// TIA Portal project "Entrega1 automatas2" (V17)

(* hardware
DEVICE "S7-1200 station_1"  S7-1200 Station
   slot 0: "Rack_0"  S7-1200 Rack  Rack  V1.0
   slot 1: "PLC_1"  CPU 1215C AC/DC/Rly  6ES7 215-1BG40-0XB0  V4.0
DEVICE "S7-1200 station_2"  S7-1200 Station
   slot 0: "Rack_0"  S7-1200 Rack  Rack  V1.0
   slot 1: "PLC_2"  CPU 1214C AC/DC/Rly  6ES7 214-1BG31-0XB0  V3.0
   slot 3: "AQ 1x12BIT_1"  AQ1 signal board  6ES7 232-4HA30-0XB0  V1.0
DEVICE "S7-1200 station_3"  S7-1200 Station
   slot 0: "Rack_0"  S7-1200 Rack  Rack  V1.0
   slot 1: "PLC_3"  CPU 1214C AC/DC/Rly  6ES7 214-1BG31-0XB0  V3.0
*)

// ===== PLC "PLC_1"  CPU 1215C AC/DC/Rly =====

VAR_GLOBAL   // PLC tag table "Default tag table"
   "i_PM" AT %I0.0 : Bool;
   "i_PP" AT %I0.1 : Bool;
   "i_FC" AT %I0.2 : Bool;
   "q_EV1" AT %Q0.0 : Bool;
   "q_EV2" AT %Q0.1 : Bool;
   "q_EV3" AT %Q0.2 : Bool;
   "q_Di1" AT %Q0.3 : Bool;
   "q_Di2" AT %Q0.4 : Bool;
   "q_Z" AT %Q0.5 : Bool;
   "q_KM1" AT %Q0.6 : Bool;
   "q_KM2" AT %Q0.7 : Bool;
   "GP_E0" AT %M50.0 : Bool;
   "GP_E1" AT %M50.1 : Bool;
   "GP_E2" AT %M50.2 : Bool;
   "GP_E3" AT %M50.3 : Bool;
   "GP_E4" AT %M50.4 : Bool;
   "GP_E5" AT %M50.5 : Bool;
   "GP_E6" AT %M50.6 : Bool;
   "GP_E7" AT %M50.7 : Bool;
   "GS_E100" AT %M51.0 : Bool;
   "GS_E101" AT %M51.1 : Bool;
   "T1" AT %MD100 : Time;
   "Minimo_distancia" AT %MD104 : Real;
   "Maximo distancia" AT %MD106 : Real;
   "Salida_Voltios" AT %MD80 : Real;
   "distancia_normalizada" AT %MD60 : Real;
   "Variable_Stop" AT %M500.0 : Bool;
END_VAR

VAR_GLOBAL   // PLC tag table "Tag table_1"
   "entrada_analogica(1)" AT %IW64 : Word;
END_VAR

// folder: System blocks/Program resources

DATA_BLOCK "T1.1"   // DB1
{ S7_Optimized_Access := 'TRUE' }
AUTHOR : Simatic
FAMILY : IEC
NAME : IEC_TMR
VERSION : 1.0
// stored: InstanceOfName IEC_TIMER
"IEC_TIMER"
BEGIN
END_DATA_BLOCK

DATA_BLOCK "T2"   // DB2
{ S7_Optimized_Access := 'TRUE' }
AUTHOR : Simatic
FAMILY : IEC
NAME : IEC_TMR
VERSION : 1.0
// stored: InstanceOfName IEC_TIMER
"IEC_TIMER"
BEGIN
END_DATA_BLOCK

DATA_BLOCK "T3"   // DB3
{ S7_Optimized_Access := 'TRUE' }
AUTHOR : Simatic
FAMILY : IEC
NAME : IEC_TMR
VERSION : 1.0
// stored: InstanceOfName IEC_TIMER
"IEC_TIMER"
BEGIN
END_DATA_BLOCK

DATA_BLOCK "T4"   // DB4
{ S7_Optimized_Access := 'TRUE' }
AUTHOR : Simatic
FAMILY : IEC
NAME : IEC_TMR
VERSION : 1.0
// stored: InstanceOfName IEC_TIMER
"IEC_TIMER"
BEGIN
END_DATA_BLOCK

// folder: (top level)

FUNCTION "Grafcet principal" : Void   // FC1, LAD
{ S7_Optimized_Access := 'TRUE' }
VERSION : 0.1
   VAR_TEMP   // added for the SCL form of the ladder/FBD networks
      _w1 : Bool;
   END_VAR
BEGIN

REGION Network 1
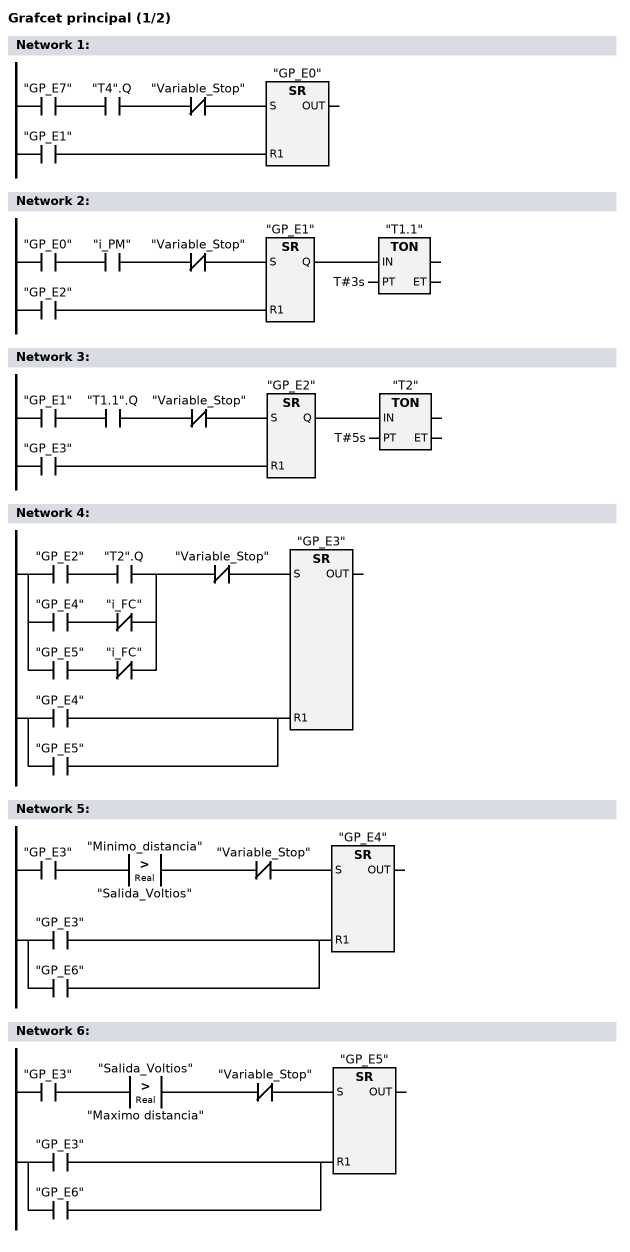
   RUNG wire#powerrail
      Contact( "GP_E7" )
      Contact( "T4".Q )
      I_Contact( "Variable_Stop" )
      S_SR(operand := "GP_E0", r1 := wire#w1)
   END_RUNG
   RUNG wire#powerrail
      Contact( "GP_E1" )
   END_RUNG wire#w1
   // the same network as SCL:
   IF "GP_E7" AND "T4".Q AND NOT "Variable_Stop" THEN
       "GP_E0" := TRUE;   // SR flip-flop
   END_IF;
   IF "GP_E1" THEN "GP_E0" := FALSE; END_IF;
END_REGION

REGION Network 2
   IF "GP_E0" AND "i_PM" AND NOT "Variable_Stop" THEN
       "GP_E1" := TRUE;   // SR flip-flop
   END_IF;
   IF "GP_E2" THEN "GP_E1" := FALSE; END_IF;
   "T1.1".TON(IN := "GP_E1", PT := T#3s);
END_REGION

REGION Network 3
   IF "GP_E1" AND "T1.1".Q AND NOT "Variable_Stop" THEN
       "GP_E2" := TRUE;   // SR flip-flop
   END_IF;
   IF "GP_E3" THEN "GP_E2" := FALSE; END_IF;
   "T2".TON(IN := "GP_E2", PT := T#5s);
END_REGION

REGION Network 4
   RUNG wire#powerrail
      Contact( "GP_E2" )
      Contact( "T2".Q )
      wire#w1
      I_Contact( "Variable_Stop" )
      S_SR(operand := "GP_E3", r1 := wire#w2)
   END_RUNG
   RUNG wire#powerrail
      Contact( "GP_E4" )
      I_Contact( "i_FC" )
   END_RUNG wire#w1
   RUNG wire#powerrail
      Contact( "GP_E5" )
      I_Contact( "i_FC" )
   END_RUNG wire#w1
   RUNG wire#powerrail
      Contact( "GP_E4" )
   END_RUNG wire#w2
   RUNG wire#powerrail
      Contact( "GP_E5" )
   END_RUNG wire#w2
   // the same network as SCL:
   IF (("GP_E2" AND "T2".Q) OR ("GP_E4" AND NOT "i_FC") OR ("GP_E5" AND NOT "i_FC")) AND NOT "Variable_Stop" THEN
       "GP_E3" := TRUE;   // SR flip-flop
   END_IF;
   IF "GP_E4" OR "GP_E5" THEN "GP_E3" := FALSE; END_IF;
END_REGION

REGION Network 5
   RUNG wire#powerrail
      Contact( "GP_E3" )
      { S7_Templates := "SrcType := Real" } GT_Contact(in1 := "Minimo_distancia", in2 := "Salida_Voltios")
      I_Contact( "Variable_Stop" )
      S_SR(operand := "GP_E4", r1 := wire#w1)
   END_RUNG
   RUNG wire#powerrail
      Contact( "GP_E3" )
   END_RUNG wire#w1
   RUNG wire#powerrail
      Contact( "GP_E6" )
   END_RUNG wire#w1
   // the same network as SCL:
   IF "GP_E3" AND ("Minimo_distancia" > "Salida_Voltios") AND NOT "Variable_Stop" THEN
       "GP_E4" := TRUE;   // SR flip-flop
   END_IF;
   IF "GP_E3" OR "GP_E6" THEN "GP_E4" := FALSE; END_IF;
END_REGION

REGION Network 6
   RUNG wire#powerrail
      Contact( "GP_E3" )
      { S7_Templates := "SrcType := Real" } GT_Contact(in1 := "Salida_Voltios", in2 := "Maximo distancia")
      I_Contact( "Variable_Stop" )
      S_SR(operand := "GP_E5", r1 := wire#w1)
   END_RUNG
   RUNG wire#powerrail
      Contact( "GP_E3" )
   END_RUNG wire#w1
   RUNG wire#powerrail
      Contact( "GP_E6" )
   END_RUNG wire#w1
   // the same network as SCL:
   IF "GP_E3" AND ("Salida_Voltios" > "Maximo distancia") AND NOT "Variable_Stop" THEN
       "GP_E5" := TRUE;   // SR flip-flop
   END_IF;
   IF "GP_E3" OR "GP_E6" THEN "GP_E5" := FALSE; END_IF;
END_REGION

REGION Network 7
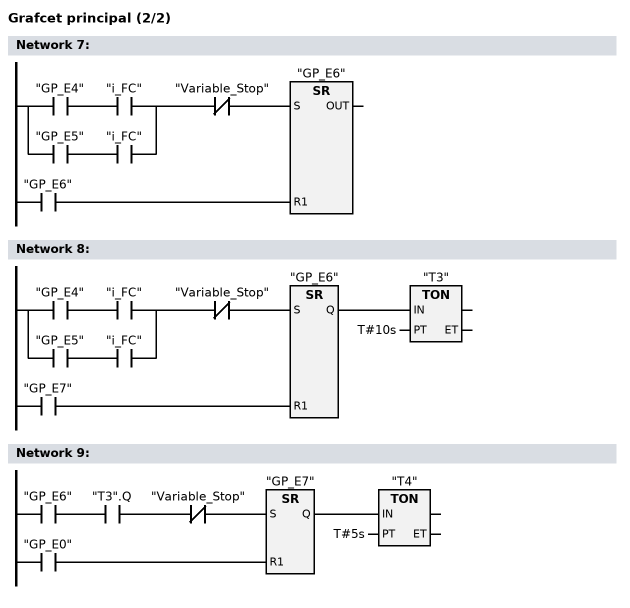
   RUNG wire#powerrail
      Contact( "GP_E4" )
      Contact( "i_FC" )
      wire#w1
      I_Contact( "Variable_Stop" )
      S_SR(operand := "GP_E6", r1 := wire#w2)
   END_RUNG
   RUNG wire#powerrail
      Contact( "GP_E5" )
      Contact( "i_FC" )
   END_RUNG wire#w1
   RUNG wire#powerrail
      Contact( "GP_E6" )
   END_RUNG wire#w2
   // the same network as SCL:
   #_w1 := "GP_E6";
   IF (("GP_E4" AND "i_FC") OR ("GP_E5" AND "i_FC")) AND NOT "Variable_Stop" THEN
       "GP_E6" := TRUE;   // SR flip-flop
   END_IF;
   IF #_w1 THEN "GP_E6" := FALSE; END_IF;
END_REGION

REGION Network 8
   IF (("GP_E4" AND "i_FC") OR ("GP_E5" AND "i_FC")) AND NOT "Variable_Stop" THEN
       "GP_E6" := TRUE;   // SR flip-flop
   END_IF;
   IF "GP_E7" THEN "GP_E6" := FALSE; END_IF;
   "T3".TON(IN := "GP_E6", PT := T#10s);
END_REGION

REGION Network 9
   IF "GP_E6" AND "T3".Q AND NOT "Variable_Stop" THEN
       "GP_E7" := TRUE;   // SR flip-flop
   END_IF;
   IF "GP_E0" THEN "GP_E7" := FALSE; END_IF;
   "T4".TON(IN := "GP_E7", PT := T#5s);
END_REGION
END_FUNCTION

FUNCTION "Grafcet Stop" : Void   // FC2, LAD
{ S7_Optimized_Access := 'TRUE' }
VERSION : 0.1
BEGIN

REGION Network 1
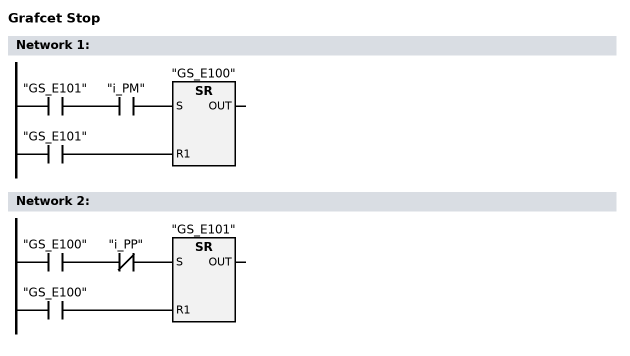
   RUNG wire#powerrail
      Contact( "GS_E101" )
      Contact( "i_PM" )
      S_SR(operand := "GS_E100", r1 := wire#w1)
   END_RUNG
   RUNG wire#powerrail
      Contact( "GS_E101" )
   END_RUNG wire#w1
   // the same network as SCL:
   IF "GS_E101" AND "i_PM" THEN
       "GS_E100" := TRUE;   // SR flip-flop
   END_IF;
   IF "GS_E101" THEN "GS_E100" := FALSE; END_IF;
END_REGION

REGION Network 2
   RUNG wire#powerrail
      Contact( "GS_E100" )
      I_Contact( "i_PP" )
      S_SR(operand := "GS_E101", r1 := wire#w1)
   END_RUNG
   RUNG wire#powerrail
      Contact( "GS_E100" )
   END_RUNG wire#w1
   // the same network as SCL:
   IF "GS_E100" AND NOT "i_PP" THEN
       "GS_E101" := TRUE;   // SR flip-flop
   END_IF;
   IF "GS_E100" THEN "GS_E101" := FALSE; END_IF;
END_REGION
END_FUNCTION

FUNCTION "Salidas" : Void   // FC3, LAD
{ S7_Optimized_Access := 'TRUE' }
VERSION : 0.1
BEGIN

REGION Network 1
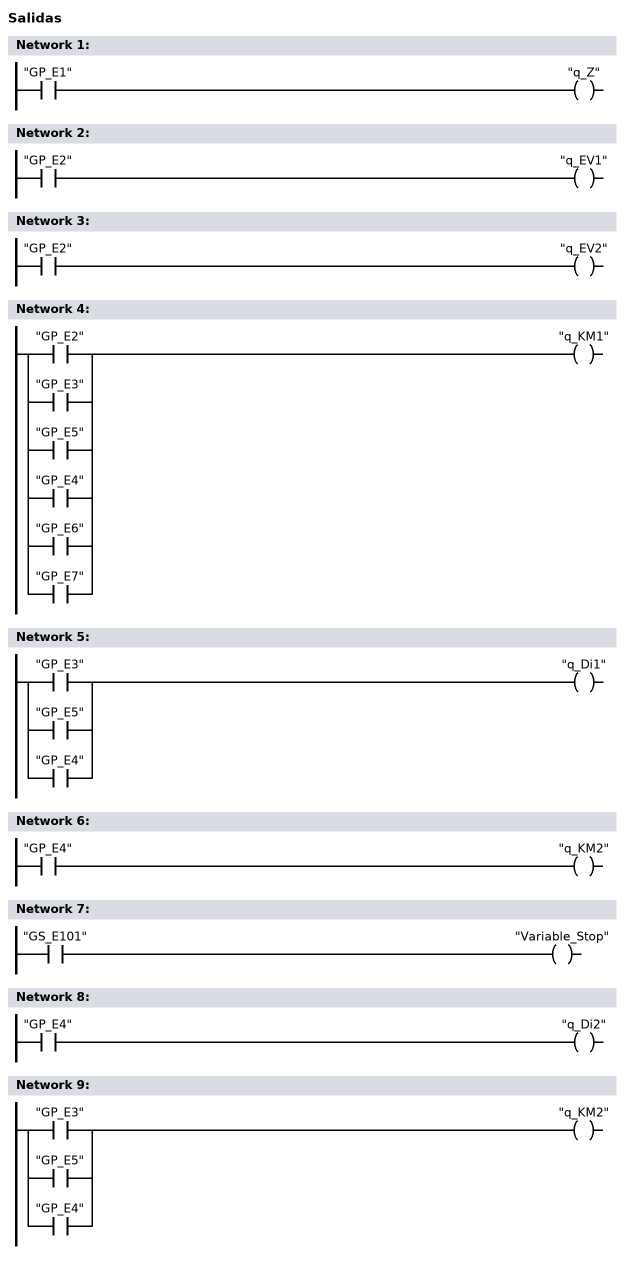
   RUNG wire#powerrail
      Contact( "GP_E1" )
      Coil( "q_Z" )
   END_RUNG
   // the same network as SCL:
   "q_Z" := "GP_E1";
END_REGION

REGION Network 2
   RUNG wire#powerrail
      Contact( "GP_E2" )
      Coil( "q_EV1" )
   END_RUNG
   // the same network as SCL:
   "q_EV1" := "GP_E2";
END_REGION

REGION Network 3
   RUNG wire#powerrail
      Contact( "GP_E2" )
      Coil( "q_EV2" )
   END_RUNG
   // the same network as SCL:
   "q_EV2" := "GP_E2";
END_REGION

REGION Network 4
   RUNG wire#powerrail
      Contact( "GP_E2" )
      wire#w1
      Coil( "q_KM1" )
   END_RUNG
   RUNG wire#powerrail
      Contact( "GP_E3" )
   END_RUNG wire#w1
   RUNG wire#powerrail
      Contact( "GP_E5" )
   END_RUNG wire#w1
   RUNG wire#powerrail
      Contact( "GP_E4" )
   END_RUNG wire#w1
   RUNG wire#powerrail
      Contact( "GP_E6" )
   END_RUNG wire#w1
   RUNG wire#powerrail
      Contact( "GP_E7" )
   END_RUNG wire#w1
   // the same network as SCL:
   "q_KM1" := "GP_E2" OR "GP_E3" OR "GP_E5" OR "GP_E4" OR "GP_E6" OR "GP_E7";
END_REGION

REGION Network 5
   RUNG wire#powerrail
      Contact( "GP_E3" )
      wire#w1
      Coil( "q_Di1" )
   END_RUNG
   RUNG wire#powerrail
      Contact( "GP_E5" )
   END_RUNG wire#w1
   RUNG wire#powerrail
      Contact( "GP_E4" )
   END_RUNG wire#w1
   // the same network as SCL:
   "q_Di1" := "GP_E3" OR "GP_E5" OR "GP_E4";
END_REGION

REGION Network 6
   RUNG wire#powerrail
      Contact( "GP_E4" )
      Coil( "q_KM2" )
   END_RUNG
   // the same network as SCL:
   "q_KM2" := "GP_E4";
END_REGION

REGION Network 7
   RUNG wire#powerrail
      Contact( "GS_E101" )
      Coil( "Variable_Stop" )
   END_RUNG
   // the same network as SCL:
   "Variable_Stop" := "GS_E101";
END_REGION

REGION Network 8
   RUNG wire#powerrail
      Contact( "GP_E4" )
      Coil( "q_Di2" )
   END_RUNG
   // the same network as SCL:
   "q_Di2" := "GP_E4";
END_REGION

REGION Network 9
   RUNG wire#powerrail
      Contact( "GP_E3" )
      wire#w1
      Coil( "q_KM2" )
   END_RUNG
   RUNG wire#powerrail
      Contact( "GP_E5" )
   END_RUNG wire#w1
   RUNG wire#powerrail
      Contact( "GP_E4" )
   END_RUNG wire#w1
   // the same network as SCL:
   "q_KM2" := "GP_E3" OR "GP_E5" OR "GP_E4";
END_REGION
END_FUNCTION

FUNCTION "Analogicas" : Void   // FC4, LAD
{ S7_Optimized_Access := 'TRUE' }
VERSION : 0.1
BEGIN

REGION Network 1
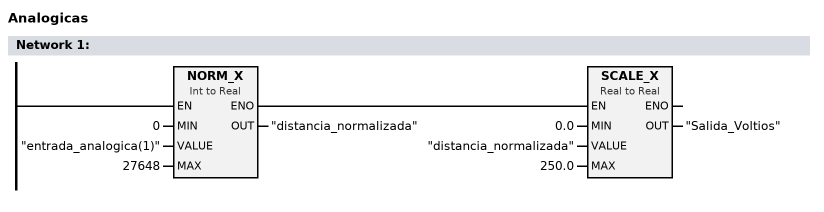
   RUNG wire#powerrail
      { S7_Templates := "[SrcType := Int, DestType := Real]" } Normalize(min := 0, value := "entrada_analogica(1)", max := 27648, out => "distancia_normalizada")
      { S7_Templates := "[SrcType := Real, DestType := Real]" } Scale(min := 0.0, value := "distancia_normalizada", max := 250.0, out => "Salida_Voltios")
   END_RUNG
   // the same network as SCL:
   "distancia_normalizada" := NORM_X(MIN := 0, VALUE := "entrada_analogica(1)", MAX := 27648);
   "Salida_Voltios" := SCALE_X(MIN := 0.0, VALUE := "distancia_normalizada", MAX := 250.0);
END_REGION
END_FUNCTION

ORGANIZATION_BLOCK "Main"   // OB1, LAD, ProgramCycle
TITLE = "Main Program Sweep (Cycle)"
{ S7_Optimized_Access := 'TRUE' }
VERSION : 0.1
   VAR_INPUT
      Initial_Call : Bool;   // Initial call of this OB
      Remanence : Bool;   // =True, if remanent data are available
   END_VAR
BEGIN

REGION Network 1
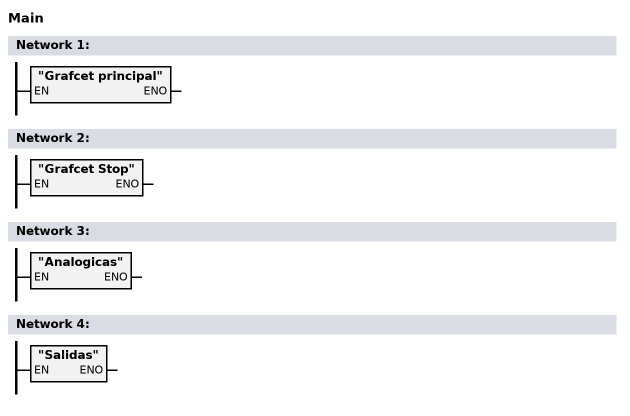
   RUNG wire#powerrail
      "Grafcet principal"()
   END_RUNG
   // the same network as SCL:
   "Grafcet principal"();
END_REGION

REGION Network 2
   RUNG wire#powerrail
      "Grafcet Stop"()
   END_RUNG
   // the same network as SCL:
   "Grafcet Stop"();
END_REGION

REGION Network 3
   RUNG wire#powerrail
      "Analogicas"()
   END_RUNG
   // the same network as SCL:
   "Analogicas"();
END_REGION

REGION Network 4
   RUNG wire#powerrail
      "Salidas"()
   END_RUNG
   // the same network as SCL:
   "Salidas"();
END_REGION
END_ORGANIZATION_BLOCK

ORGANIZATION_BLOCK "Startup"   // OB100, LAD, Startup
TITLE = "Complete Restart"
{ S7_Optimized_Access := 'TRUE' }
VERSION : 0.1
   VAR_INPUT
      LostRetentive : Bool;   // True if retentive data are lost
      LostRTC : Bool;   // True if date and time are lost
   END_VAR
BEGIN

REGION Network 1
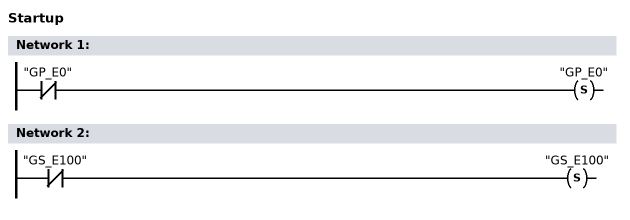
   RUNG wire#powerrail
      I_Contact( "GP_E0" )
      S_Coil( "GP_E0" )
   END_RUNG
   // the same network as SCL:
   IF NOT "GP_E0" THEN "GP_E0" := TRUE; END_IF;
END_REGION

REGION Network 2
   RUNG wire#powerrail
      I_Contact( "GS_E100" )
      S_Coil( "GS_E100" )
   END_RUNG
   // the same network as SCL:
   IF NOT "GS_E100" THEN "GS_E100" := TRUE; END_IF;
END_REGION
END_ORGANIZATION_BLOCK

// ===== PLC "PLC_2"  CPU 1214C AC/DC/Rly =====

VAR_GLOBAL   // PLC tag table "Default tag table"
   "GP_E4.5" AT %M51.2 : Bool;
   "Tag_1" AT %MB800 : Byte;
END_VAR

VAR_GLOBAL   // PLC tag table "Default tag table_1"
   "i_PM" AT %I0.0 : Bool;
   "i_PP" AT %I0.1 : Bool;
   "i_FC" AT %I0.2 : Bool;
   "q_EV1" AT %Q0.0 : Bool;
   "q_EV2" AT %Q0.1 : Bool;
   "q_EV3" AT %Q0.2 : Bool;
   "q_Di1" AT %Q0.3 : Bool;
   "q_Di2" AT %Q0.4 : Bool;
   "q_Z" AT %Q0.5 : Bool;
   "q_KM1" AT %Q0.6 : Bool;
   "q_KM2" AT %Q0.7 : Bool;
   "GP_E0" AT %M50.0 : Bool;
   "GP_E1" AT %M50.1 : Bool;
   "GP_E2" AT %M50.2 : Bool;
   "GP_E3" AT %M50.3 : Bool;
   "GP_E4" AT %M50.4 : Bool;
   "GP_E5" AT %M50.5 : Bool;
   "GP_E6" AT %M50.6 : Bool;
   "GP_E7" AT %M50.7 : Bool;
   "GS_E100" AT %M51.0 : Bool;
   "GS_E101" AT %M51.1 : Bool;
   "T1" AT %MD100 : Time;
   "Minimo_distancia" AT %MD104 : Real;
   "Maximo distancia" AT %MD106 : Real;
   "Salida_Voltios" AT %MD80 : Real;
   "distancia_normalizada" AT %MD60 : Real;
   "Variable_Stop" AT %M500.0 : Bool;
   "velocidad_hz" AT %MD108 : Real;
   "velocidad_normalizada" AT %MD112 : Real;
   "salida_velocidad" AT %QW80 : Int;
   "GP_E8" AT %M51.3 : Bool;
END_VAR

VAR_GLOBAL CONSTANT   // PLC tag table "Default tag table_1"
   "None" : Pip := 65535;
   "Automatic update" : Pip := 0;
   "PIP 1" : Pip := 1;
   "PIP 2" : Pip := 2;
   "PIP 3" : Pip := 3;
   "PIP 4" : Pip := 4;
   "PIP OB Servo" : Pip := 32768;
   "Local~MC" : Hw_SubModule := 51;
   "Local~Common" : Hw_SubModule := 50;
   "Local~Exec" : Hw_SubModule := 52;
   "Local(1)" : Hw_SubModule := 49;
   "Local~PROFINET_interface_1(1)" : Hw_Interface := 64;
   "Local~PROFINET_interface_1~Port_1(1)" : Hw_Interface := 65;
   "Local~PROFINET_interface_1~Port_2" : Hw_Interface := 66;
   "Local~HSC_1(1)" : Hw_Hsc := 257;
   "Local~HSC_2(1)" : Hw_Hsc := 258;
   "Local~HSC_3(1)" : Hw_Hsc := 259;
   "Local~HSC_4(1)" : Hw_Hsc := 260;
   "Local~HSC_5(1)" : Hw_Hsc := 261;
   "Local~HSC_6(1)" : Hw_Hsc := 262;
   "Local~AI_2_AQ_2_1" : Hw_SubModule := 263;
   "Local~DI_14_DQ_10_1(1)" : Hw_SubModule := 264;
   "Local~Pulse_1(1)" : Hw_Pwm := 265;
   "Local~Pulse_2(1)" : Hw_Pwm := 266;
   "Local~Pulse_3(1)" : Hw_Pwm := 267;
   "Local~Pulse_4(1)" : Hw_Pwm := 268;
   "OB_Main(1)" : OB_PCYCLE := 1;
   "OB_Startup(1)" : OB_STARTUP := 100;
END_VAR

VAR_GLOBAL   // PLC tag table "Tag table_1"
   "entrada_analogica(1)" AT %IW64 : Word;
   "flanco1" AT %M2.0 : Bool;
   "flanco2" AT %M3.0 : Bool;
   "flanco3" AT %M4.0 : Bool;
   "flanco4" AT %M4.1 : Bool;
   "flanco5" AT %M4.2 : Bool;
   "flanco6" AT %M4.3 : Bool;
   "flanco7" AT %M4.4 : Bool;
   "flanco8" AT %M4.5 : Bool;
   "salida_hz" AT %MD84 : Real;
   "flanco9" AT %M4.6 : Bool;
END_VAR

// folder: System blocks/Program resources

DATA_BLOCK "T1.1"   // DB1
{ S7_Optimized_Access := 'TRUE' }
AUTHOR : Simatic
FAMILY : IEC
NAME : IEC_TMR
VERSION : 1.0
// stored: InstanceOfName IEC_TIMER
"IEC_TIMER"
BEGIN
END_DATA_BLOCK

DATA_BLOCK "T2"   // DB2
{ S7_Optimized_Access := 'TRUE' }
AUTHOR : Simatic
FAMILY : IEC
NAME : IEC_TMR
VERSION : 1.0
// stored: InstanceOfName IEC_TIMER
"IEC_TIMER"
BEGIN
END_DATA_BLOCK

DATA_BLOCK "T3"   // DB3
{ S7_Optimized_Access := 'TRUE' }
AUTHOR : Simatic
FAMILY : IEC
NAME : IEC_TMR
VERSION : 1.0
// stored: InstanceOfName IEC_TIMER
"IEC_TIMER"
BEGIN
END_DATA_BLOCK

DATA_BLOCK "T4"   // DB4
{ S7_Optimized_Access := 'TRUE' }
AUTHOR : Simatic
FAMILY : IEC
NAME : IEC_TMR
VERSION : 1.0
// stored: InstanceOfName IEC_TIMER
"IEC_TIMER"
BEGIN
END_DATA_BLOCK

// folder: (top level)

FUNCTION "Grafcet principal" : Void   // FC1, LAD
{ S7_Optimized_Access := 'TRUE' }
VERSION : 0.1
   VAR_TEMP   // added for the SCL form of the ladder/FBD networks
      _w1 : Bool;
      _w2 : Bool;
      _w3 : Bool;
   END_VAR
BEGIN

REGION Network 1
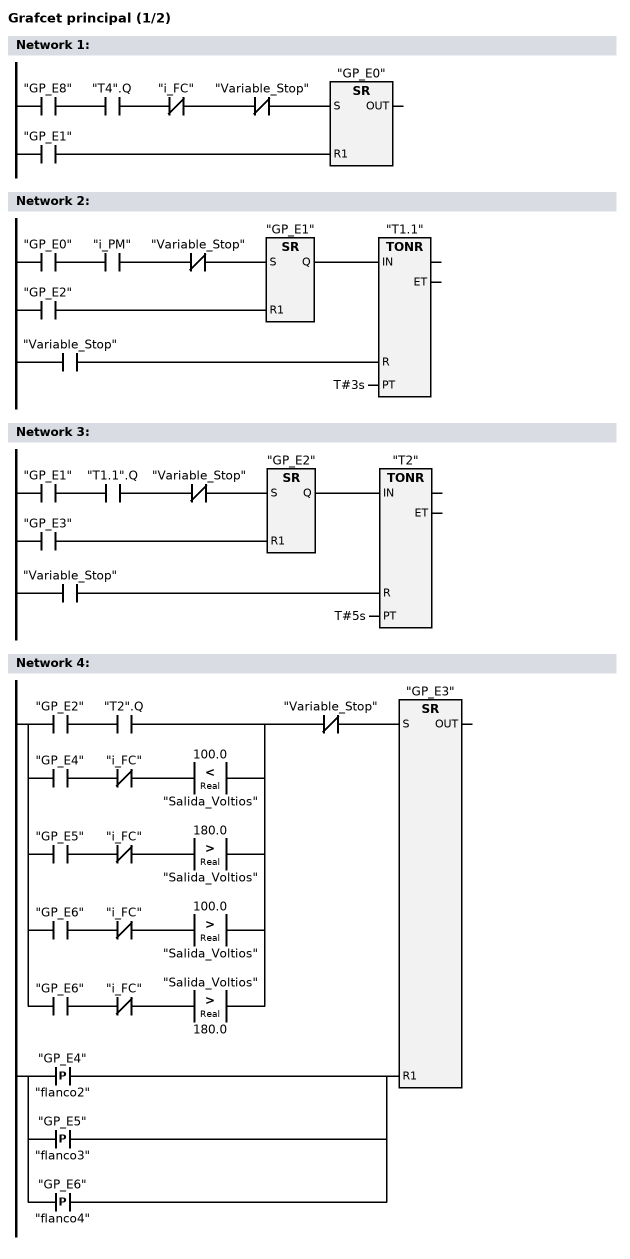
   RUNG wire#powerrail
      Contact( "GP_E8" )
      Contact( "T4".Q )
      I_Contact( "i_FC" )
      I_Contact( "Variable_Stop" )
      S_SR(operand := "GP_E0", r1 := wire#w1)
   END_RUNG
   RUNG wire#powerrail
      Contact( "GP_E1" )
   END_RUNG wire#w1
   // the same network as SCL:
   IF "GP_E8" AND "T4".Q AND NOT "i_FC" AND NOT "Variable_Stop" THEN
       "GP_E0" := TRUE;   // SR flip-flop
   END_IF;
   IF "GP_E1" THEN "GP_E0" := FALSE; END_IF;
END_REGION

REGION Network 2
   IF "GP_E0" AND "i_PM" AND NOT "Variable_Stop" THEN
       "GP_E1" := TRUE;   // SR flip-flop
   END_IF;
   IF "GP_E2" THEN "GP_E1" := FALSE; END_IF;
   "T1.1".TONR(IN := "GP_E1", R := "Variable_Stop", PT := T#3s);
END_REGION

REGION Network 3
   IF "GP_E1" AND "T1.1".Q AND NOT "Variable_Stop" THEN
       "GP_E2" := TRUE;   // SR flip-flop
   END_IF;
   IF "GP_E3" THEN "GP_E2" := FALSE; END_IF;
   "T2".TONR(IN := "GP_E2", R := "Variable_Stop", PT := T#5s);
END_REGION

REGION Network 4
   RUNG wire#powerrail
      Contact( "GP_E2" )
      Contact( "T2".Q )
      wire#w1
      I_Contact( "Variable_Stop" )
      S_SR(operand := "GP_E3", r1 := wire#w2)
   END_RUNG
   RUNG wire#powerrail
      Contact( "GP_E4" )
      I_Contact( "i_FC" )
      { S7_Templates := "SrcType := Real" } LT_Contact(in1 := 100.0, in2 := "Salida_Voltios")
   END_RUNG wire#w1
   RUNG wire#powerrail
      Contact( "GP_E5" )
      I_Contact( "i_FC" )
      { S7_Templates := "SrcType := Real" } GT_Contact(in1 := 180.0, in2 := "Salida_Voltios")
   END_RUNG wire#w1
   RUNG wire#powerrail
      Contact( "GP_E6" )
      I_Contact( "i_FC" )
      { S7_Templates := "SrcType := Real" } GT_Contact(in1 := 100.0, in2 := "Salida_Voltios")
   END_RUNG wire#w1
   RUNG wire#powerrail
      Contact( "GP_E6" )
      I_Contact( "i_FC" )
      { S7_Templates := "SrcType := Real" } GT_Contact(in1 := "Salida_Voltios", in2 := 180.0)
   END_RUNG wire#w1
   RUNG wire#powerrail
      P_Contact(operand := "GP_E4", bit := "flanco2")
   END_RUNG wire#w2
   RUNG wire#powerrail
      P_Contact(operand := "GP_E5", bit := "flanco3")
   END_RUNG wire#w2
   RUNG wire#powerrail
      P_Contact(operand := "GP_E6", bit := "flanco4")
   END_RUNG wire#w2
   // the same network as SCL:
   #_w1 := "GP_E4" AND NOT "flanco2";   // rising edge of "GP_E4"
   "flanco2" := "GP_E4";
   #_w2 := "GP_E5" AND NOT "flanco3";   // rising edge of "GP_E5"
   "flanco3" := "GP_E5";
   #_w3 := "GP_E6" AND NOT "flanco4";   // rising edge of "GP_E6"
   "flanco4" := "GP_E6";
   IF (("GP_E2" AND "T2".Q) OR ("GP_E4" AND NOT "i_FC" AND (100.0 < "Salida_Voltios")) OR ("GP_E5" AND NOT "i_FC" AND (180.0 > "Salida_Voltios")) OR ("GP_E6" AND NOT "i_FC" AND (100.0 > "Salida_Voltios")) OR ("GP_E6" AND NOT "i_FC" AND ("Salida_Voltios" > 180.0))) AND NOT "Variable_Stop" THEN
       "GP_E3" := TRUE;   // SR flip-flop
   END_IF;
   IF #_w1 OR #_w2 OR #_w3 THEN "GP_E3" := FALSE; END_IF;
END_REGION

REGION Network 5
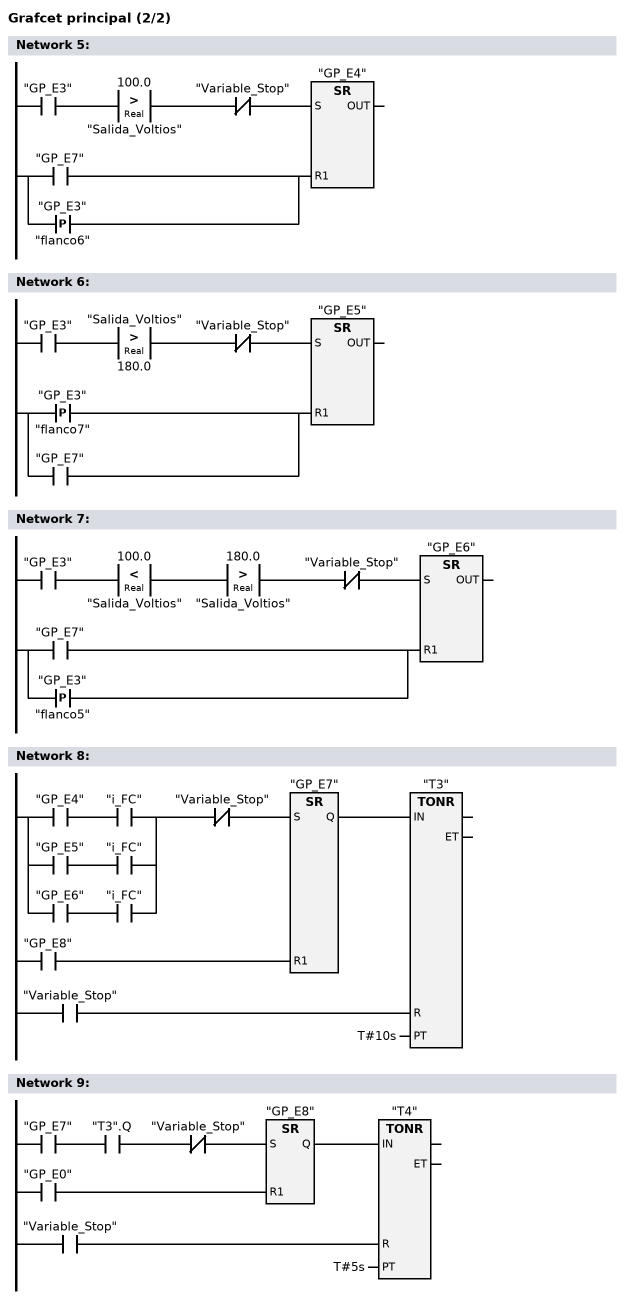
   RUNG wire#powerrail
      Contact( "GP_E3" )
      { S7_Templates := "SrcType := Real" } GT_Contact(in1 := 100.0, in2 := "Salida_Voltios")
      I_Contact( "Variable_Stop" )
      S_SR(operand := "GP_E4", r1 := wire#w1)
   END_RUNG
   RUNG wire#powerrail
      Contact( "GP_E7" )
   END_RUNG wire#w1
   RUNG wire#powerrail
      P_Contact(operand := "GP_E3", bit := "flanco6")
   END_RUNG wire#w1
   // the same network as SCL:
   #_w1 := "GP_E3" AND NOT "flanco6";   // rising edge of "GP_E3"
   "flanco6" := "GP_E3";
   IF "GP_E3" AND (100.0 > "Salida_Voltios") AND NOT "Variable_Stop" THEN
       "GP_E4" := TRUE;   // SR flip-flop
   END_IF;
   IF "GP_E7" OR #_w1 THEN "GP_E4" := FALSE; END_IF;
END_REGION

REGION Network 6
   RUNG wire#powerrail
      Contact( "GP_E3" )
      { S7_Templates := "SrcType := Real" } GT_Contact(in1 := "Salida_Voltios", in2 := 180.0)
      I_Contact( "Variable_Stop" )
      S_SR(operand := "GP_E5", r1 := wire#w1)
   END_RUNG
   RUNG wire#powerrail
      P_Contact(operand := "GP_E3", bit := "flanco7")
   END_RUNG wire#w1
   RUNG wire#powerrail
      Contact( "GP_E7" )
   END_RUNG wire#w1
   // the same network as SCL:
   #_w1 := "GP_E3" AND NOT "flanco7";   // rising edge of "GP_E3"
   "flanco7" := "GP_E3";
   IF "GP_E3" AND ("Salida_Voltios" > 180.0) AND NOT "Variable_Stop" THEN
       "GP_E5" := TRUE;   // SR flip-flop
   END_IF;
   IF #_w1 OR "GP_E7" THEN "GP_E5" := FALSE; END_IF;
END_REGION

REGION Network 7
   RUNG wire#powerrail
      Contact( "GP_E3" )
      { S7_Templates := "SrcType := Real" } LT_Contact(in1 := 100.0, in2 := "Salida_Voltios")
      { S7_Templates := "SrcType := Real" } GT_Contact(in1 := 180.0, in2 := "Salida_Voltios")
      I_Contact( "Variable_Stop" )
      S_SR(operand := "GP_E6", r1 := wire#w1)
   END_RUNG
   RUNG wire#powerrail
      Contact( "GP_E7" )
   END_RUNG wire#w1
   RUNG wire#powerrail
      P_Contact(operand := "GP_E3", bit := "flanco5")
   END_RUNG wire#w1
   // the same network as SCL:
   #_w1 := "GP_E3" AND NOT "flanco5";   // rising edge of "GP_E3"
   "flanco5" := "GP_E3";
   IF "GP_E3" AND (100.0 < "Salida_Voltios") AND (180.0 > "Salida_Voltios") AND NOT "Variable_Stop" THEN
       "GP_E6" := TRUE;   // SR flip-flop
   END_IF;
   IF "GP_E7" OR #_w1 THEN "GP_E6" := FALSE; END_IF;
END_REGION

REGION Network 8
   IF (("GP_E4" AND "i_FC") OR ("GP_E5" AND "i_FC") OR ("GP_E6" AND "i_FC")) AND NOT "Variable_Stop" THEN
       "GP_E7" := TRUE;   // SR flip-flop
   END_IF;
   IF "GP_E8" THEN "GP_E7" := FALSE; END_IF;
   "T3".TONR(IN := "GP_E7", R := "Variable_Stop", PT := T#10s);
END_REGION

REGION Network 9
   IF "GP_E7" AND "T3".Q AND NOT "Variable_Stop" THEN
       "GP_E8" := TRUE;   // SR flip-flop
   END_IF;
   IF "GP_E0" THEN "GP_E8" := FALSE; END_IF;
   "T4".TONR(IN := "GP_E8", R := "Variable_Stop", PT := T#5s);
END_REGION
END_FUNCTION

FUNCTION "Grafcet Stop" : Void   // FC2, LAD
{ S7_Optimized_Access := 'TRUE' }
VERSION : 0.1
   VAR_TEMP   // added for the SCL form of the ladder/FBD networks
      _w1 : Bool;
   END_VAR
BEGIN

REGION Network 1
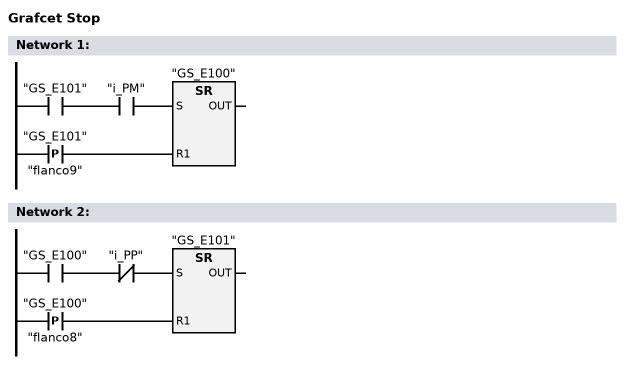
   RUNG wire#powerrail
      Contact( "GS_E101" )
      Contact( "i_PM" )
      S_SR(operand := "GS_E100", r1 := wire#w1)
   END_RUNG
   RUNG wire#powerrail
      P_Contact(operand := "GS_E101", bit := "flanco9")
   END_RUNG wire#w1
   // the same network as SCL:
   #_w1 := "GS_E101" AND NOT "flanco9";   // rising edge of "GS_E101"
   "flanco9" := "GS_E101";
   IF "GS_E101" AND "i_PM" THEN
       "GS_E100" := TRUE;   // SR flip-flop
   END_IF;
   IF #_w1 THEN "GS_E100" := FALSE; END_IF;
END_REGION

REGION Network 2
   RUNG wire#powerrail
      Contact( "GS_E100" )
      I_Contact( "i_PP" )
      S_SR(operand := "GS_E101", r1 := wire#w1)
   END_RUNG
   RUNG wire#powerrail
      P_Contact(operand := "GS_E100", bit := "flanco8")
   END_RUNG wire#w1
   // the same network as SCL:
   #_w1 := "GS_E100" AND NOT "flanco8";   // rising edge of "GS_E100"
   "flanco8" := "GS_E100";
   IF "GS_E100" AND NOT "i_PP" THEN
       "GS_E101" := TRUE;   // SR flip-flop
   END_IF;
   IF #_w1 THEN "GS_E101" := FALSE; END_IF;
END_REGION
END_FUNCTION

FUNCTION "Salidas" : Void   // FC3, LAD
{ S7_Optimized_Access := 'TRUE' }
VERSION : 0.1
BEGIN

REGION Network 1
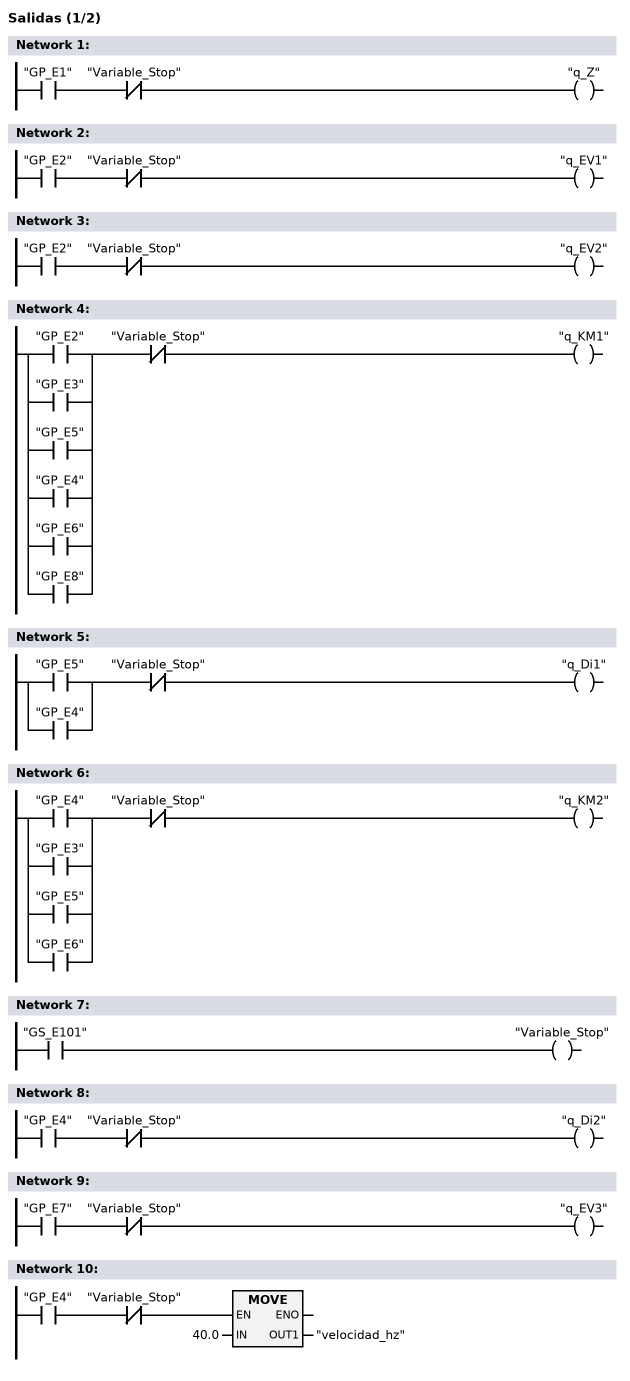
   RUNG wire#powerrail
      Contact( "GP_E1" )
      I_Contact( "Variable_Stop" )
      Coil( "q_Z" )
   END_RUNG
   // the same network as SCL:
   "q_Z" := "GP_E1" AND NOT "Variable_Stop";
END_REGION

REGION Network 2
   RUNG wire#powerrail
      Contact( "GP_E2" )
      I_Contact( "Variable_Stop" )
      Coil( "q_EV1" )
   END_RUNG
   // the same network as SCL:
   "q_EV1" := "GP_E2" AND NOT "Variable_Stop";
END_REGION

REGION Network 3
   RUNG wire#powerrail
      Contact( "GP_E2" )
      I_Contact( "Variable_Stop" )
      Coil( "q_EV2" )
   END_RUNG
   // the same network as SCL:
   "q_EV2" := "GP_E2" AND NOT "Variable_Stop";
END_REGION

REGION Network 4
   RUNG wire#powerrail
      Contact( "GP_E2" )
      wire#w1
      I_Contact( "Variable_Stop" )
      Coil( "q_KM1" )
   END_RUNG
   RUNG wire#powerrail
      Contact( "GP_E3" )
   END_RUNG wire#w1
   RUNG wire#powerrail
      Contact( "GP_E5" )
   END_RUNG wire#w1
   RUNG wire#powerrail
      Contact( "GP_E4" )
   END_RUNG wire#w1
   RUNG wire#powerrail
      Contact( "GP_E6" )
   END_RUNG wire#w1
   RUNG wire#powerrail
      Contact( "GP_E8" )
   END_RUNG wire#w1
   // the same network as SCL:
   "q_KM1" := ("GP_E2" OR "GP_E3" OR "GP_E5" OR "GP_E4" OR "GP_E6" OR "GP_E8") AND NOT "Variable_Stop";
END_REGION

REGION Network 5
   RUNG wire#powerrail
      Contact( "GP_E5" )
      wire#w1
      I_Contact( "Variable_Stop" )
      Coil( "q_Di1" )
   END_RUNG
   RUNG wire#powerrail
      Contact( "GP_E4" )
   END_RUNG wire#w1
   // the same network as SCL:
   "q_Di1" := ("GP_E5" OR "GP_E4") AND NOT "Variable_Stop";
END_REGION

REGION Network 6
   RUNG wire#powerrail
      Contact( "GP_E4" )
      wire#w1
      I_Contact( "Variable_Stop" )
      Coil( "q_KM2" )
   END_RUNG
   RUNG wire#powerrail
      Contact( "GP_E3" )
   END_RUNG wire#w1
   RUNG wire#powerrail
      Contact( "GP_E5" )
   END_RUNG wire#w1
   RUNG wire#powerrail
      Contact( "GP_E6" )
   END_RUNG wire#w1
   // the same network as SCL:
   "q_KM2" := ("GP_E4" OR "GP_E3" OR "GP_E5" OR "GP_E6") AND NOT "Variable_Stop";
END_REGION

REGION Network 7
   RUNG wire#powerrail
      Contact( "GS_E101" )
      Coil( "Variable_Stop" )
   END_RUNG
   // the same network as SCL:
   "Variable_Stop" := "GS_E101";
END_REGION

REGION Network 8
   RUNG wire#powerrail
      Contact( "GP_E4" )
      I_Contact( "Variable_Stop" )
      Coil( "q_Di2" )
   END_RUNG
   // the same network as SCL:
   "q_Di2" := "GP_E4" AND NOT "Variable_Stop";
END_REGION

REGION Network 9
   RUNG wire#powerrail
      Contact( "GP_E7" )
      I_Contact( "Variable_Stop" )
      Coil( "q_EV3" )
   END_RUNG
   // the same network as SCL:
   "q_EV3" := "GP_E7" AND NOT "Variable_Stop";
END_REGION

REGION Network 10
   RUNG wire#powerrail
      Contact( "GP_E4" )
      I_Contact( "Variable_Stop" )
      { S7_GenerateENO := "TRUE" } Move(in := 40.0, out1 => "velocidad_hz")
   END_RUNG
   // the same network as SCL:
   IF "GP_E4" AND NOT "Variable_Stop" THEN "velocidad_hz" := 40.0; END_IF;
END_REGION

REGION Network 11
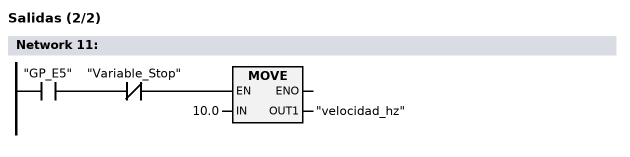
   RUNG wire#powerrail
      Contact( "GP_E5" )
      I_Contact( "Variable_Stop" )
      { S7_GenerateENO := "TRUE" } Move(in := 10.0, out1 => "velocidad_hz")
   END_RUNG
   // the same network as SCL:
   IF "GP_E5" AND NOT "Variable_Stop" THEN "velocidad_hz" := 10.0; END_IF;
END_REGION
END_FUNCTION

FUNCTION "Analogicas" : Void   // FC4, LAD
{ S7_Optimized_Access := 'TRUE' }
VERSION : 0.1
BEGIN

REGION Network 1
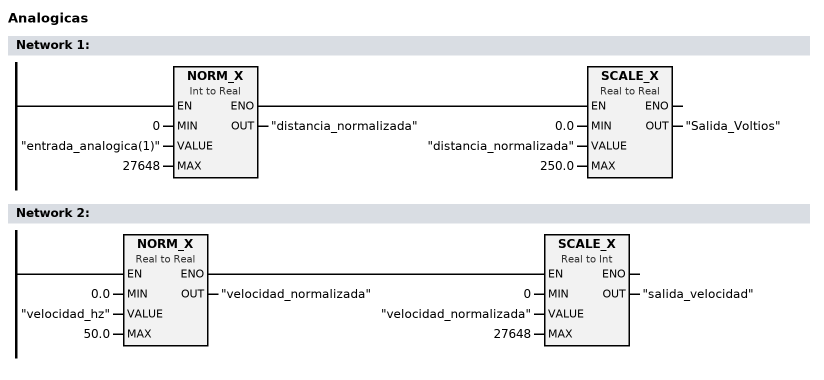
   RUNG wire#powerrail
      { S7_Templates := "[SrcType := Int, DestType := Real]"; S7_GenerateENO := "TRUE" } Normalize(min := 0, value := "entrada_analogica(1)", max := 27648, out => "distancia_normalizada")
      { S7_Templates := "[SrcType := Real, DestType := Real]"; S7_GenerateENO := "TRUE" } Scale(min := 0.0, value := "distancia_normalizada", max := 250.0, out => "Salida_Voltios")
   END_RUNG
   // the same network as SCL:
   // ENO of a box is taken as its EN; it also drops when the box reports an error
   "distancia_normalizada" := NORM_X(MIN := 0, VALUE := "entrada_analogica(1)", MAX := 27648);
   "Salida_Voltios" := SCALE_X(MIN := 0.0, VALUE := "distancia_normalizada", MAX := 250.0);
END_REGION

REGION Network 2
   RUNG wire#powerrail
      { S7_Templates := "[SrcType := Real, DestType := Real]"; S7_GenerateENO := "TRUE" } Normalize(min := 0.0, value := "velocidad_hz", max := 50.0, out => "velocidad_normalizada")
      { S7_Templates := "[SrcType := Real, DestType := Int]"; S7_GenerateENO := "TRUE" } Scale(min := 0, value := "velocidad_normalizada", max := 27648, out => "salida_velocidad")
   END_RUNG
   // the same network as SCL:
   // ENO of a box is taken as its EN; it also drops when the box reports an error
   "velocidad_normalizada" := NORM_X(MIN := 0.0, VALUE := "velocidad_hz", MAX := 50.0);
   "salida_velocidad" := SCALE_X(MIN := 0, VALUE := "velocidad_normalizada", MAX := 27648);
END_REGION
END_FUNCTION

ORGANIZATION_BLOCK "Main"   // OB1, LAD, ProgramCycle
TITLE = "Main Program Sweep (Cycle)"
{ S7_Optimized_Access := 'TRUE' }
VERSION : 0.1
   VAR_INPUT
      Initial_Call : Bool;   // Initial call of this OB
      Remanence : Bool;   // =True, if remanent data are available
   END_VAR
BEGIN

REGION Network 1
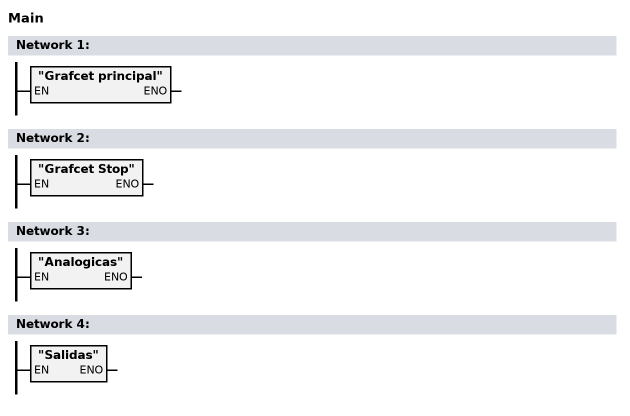
   RUNG wire#powerrail
      "Grafcet principal"()
   END_RUNG
   // the same network as SCL:
   "Grafcet principal"();
END_REGION

REGION Network 2
   RUNG wire#powerrail
      "Grafcet Stop"()
   END_RUNG
   // the same network as SCL:
   "Grafcet Stop"();
END_REGION

REGION Network 3
   RUNG wire#powerrail
      "Analogicas"()
   END_RUNG
   // the same network as SCL:
   "Analogicas"();
END_REGION

REGION Network 4
   RUNG wire#powerrail
      "Salidas"()
   END_RUNG
   // the same network as SCL:
   "Salidas"();
END_REGION
END_ORGANIZATION_BLOCK

ORGANIZATION_BLOCK "Startup"   // OB100, LAD, Startup
TITLE = "Complete Restart"
{ S7_Optimized_Access := 'TRUE' }
VERSION : 0.1
   VAR_INPUT
      LostRetentive : Bool;   // True if retentive data are lost
      LostRTC : Bool;   // True if date and time are lost
   END_VAR
BEGIN

REGION Network 1
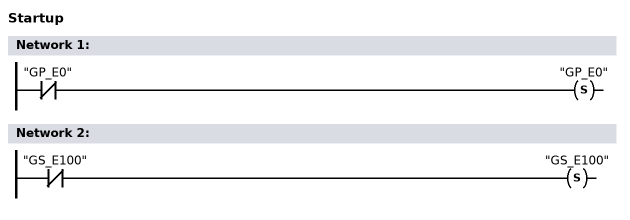
   RUNG wire#powerrail
      I_Contact( "GP_E0" )
      S_Coil( "GP_E0" )
   END_RUNG
   // the same network as SCL:
   IF NOT "GP_E0" THEN "GP_E0" := TRUE; END_IF;
END_REGION

REGION Network 2
   RUNG wire#powerrail
      I_Contact( "GS_E100" )
      S_Coil( "GS_E100" )
   END_RUNG
   // the same network as SCL:
   IF NOT "GS_E100" THEN "GS_E100" := TRUE; END_IF;
END_REGION
END_ORGANIZATION_BLOCK

// ===== PLC "PLC_3"  CPU 1214C AC/DC/Rly =====

VAR_GLOBAL   // PLC tag table "Default tag table"
   "Tag_1" AT %I0.0 : Bool;
   "Tag_2" AT %Q0.0 : Bool;
   "Tag_3" AT %Q0.1 : Bool;
   "Tag_4" AT %Q0.5 : Bool;
   "Tag_5" AT %Q0.3 : Bool;
   "Tag_6" AT %Q0.4 : Bool;
   "Tag_7" AT %MD100 : Real;
   "Tag_8" AT %MD50 : Real;
   "Tag_9" AT %IW80 : Int;
END_VAR

ORGANIZATION_BLOCK "Main"   // OB1, LAD, ProgramCycle
TITLE = "Main Program Sweep (Cycle)"
{ S7_Optimized_Access := 'TRUE' }
VERSION : 0.1
BEGIN

REGION Network 1
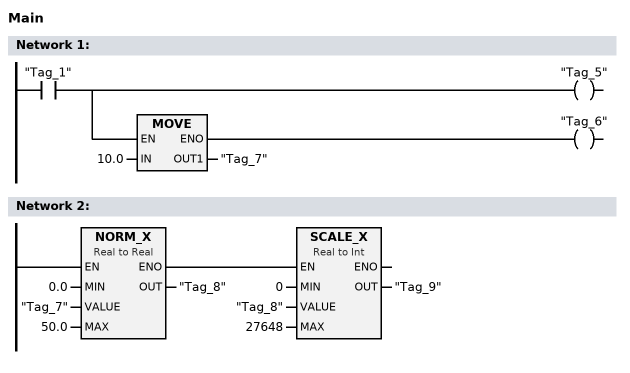
   RUNG wire#powerrail
      Contact( "Tag_1" )
      wire#w1
      Coil( "Tag_5" )
   END_RUNG
   RUNG wire#w1
      { S7_GenerateENO := "TRUE" } Move(in := 10.0, out1 => "Tag_7")
      Coil( "Tag_6" )
   END_RUNG
   // the same network as SCL:
   // ENO of a box is taken as its EN; it also drops when the box reports an error
   "Tag_5" := "Tag_1";
   IF "Tag_1" THEN "Tag_7" := 10.0; END_IF;
   "Tag_6" := "Tag_1";
END_REGION

REGION Network 2
   RUNG wire#powerrail
      { S7_Templates := "[SrcType := Real, DestType := Real]"; S7_GenerateENO := "TRUE" } Normalize(min := 0.0, value := "Tag_7", max := 50.0, out => "Tag_8")
      { S7_Templates := "[SrcType := Real, DestType := Int]"; S7_GenerateENO := "TRUE" } Scale(min := 0, value := "Tag_8", max := 27648, out => "Tag_9")
   END_RUNG
   // the same network as SCL:
   // ENO of a box is taken as its EN; it also drops when the box reports an error
   "Tag_8" := NORM_X(MIN := 0.0, VALUE := "Tag_7", MAX := 50.0);
   "Tag_9" := SCALE_X(MIN := 0, VALUE := "Tag_8", MAX := 27648);
END_REGION
END_ORGANIZATION_BLOCK